(* PLC project Unnamed, Unknown Unnamed 1 *)
(* stored: creationDateTime 2023-03-15T11:48:28, modificationDateTime 2023-03-30T09:56:05 *)

TYPE datatype0 : BOOL;
END_TYPE

PROGRAM FactoryIOtest
  VAR
    I_Start AT %IX100.0 : BOOL;
    I_Stop AT %IX100.1 : BOOL;
    Q_Conveyor AT %QX100.0 : BOOL;
  END_VAR

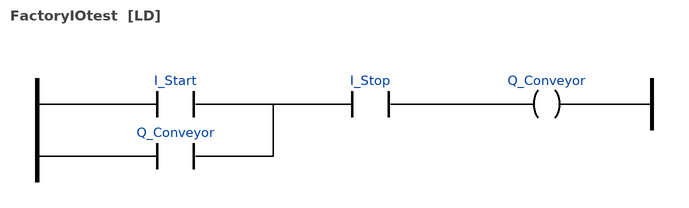
(* LD diagram, written out as Structured Text *)
Q_Conveyor := (I_Start OR Q_Conveyor) AND I_Stop;
END_PROGRAM

CONFIGURATION Config0
  RESOURCE Res0 ON PLC
    TASK task0(INTERVAL := T#20ms, PRIORITY := 0);
    PROGRAM instance0 WITH task0 : FactoryIOtest;
  END_RESOURCE
END_CONFIGURATION
